{attribute 'reflection'} 
// Providing the event logger
FUNCTION_BLOCK FB_Event IMPLEMENTS I_Event
VAR_INPUT
	iLogger:					I_Logger;		// Interface has to be attached to a Valid target
END_VAR
VAR
    {attribute 'hide'} 
    {attribute 'instance-path'} 
    {attribute 'noinit'} 
    sInstancePath:				STRING(255);
	fbSymbolInfo: 				PLC_ReadSymInfoByNameEx;
	fbSystemTime: 				FB_LocalSystemTime;
	fbArguments:				FB_Argument;	
	fbVerbose:					FB_Message;
	fbInfo:						FB_Message;
	fbWarning:					FB_Message;
	fbError:					FB_Message;
	fbCritical:					FB_Message;
END_VAR
VAR_STAT
	nCycleTime:					UDINT;
	nTimestamp:					Tc2_Utilities.T_FILETIME64;		
END_VAR
(*
    Tc3_Event – TwinCAT 3 Event Logging Framework
    Copyright (c) Peter Zerlauth

    This component is provided under a Dual Licensing Model:

    1. GPLv3 Open-Source License
       - Free for personal, educational, and non-commercial use.
       - Commercial use allowed only if the entire application is published
         under GPLv3, including all modifications to this code.
       - Requires full disclosure of source code for derivative works.

    2. Commercial License
       - Required for integration into proprietary or closed-source products.
       - Removes all GPLv3 copyleft obligations.
       - Includes optional warranty, professional support, and long-term
         maintenance options.

    For commercial licensing, contact:
        info@peterzerlauth.com

    By using this Function Block you agree to the terms of the selected license.
*)

fbSymbolInfo();
IF nCycleTime <> TwinCAT_SystemInfoVarList._TaskInfo[GETCURTASKINDEXEX()].CycleTime THEN
	nCycleTime:= TwinCAT_SystemInfoVarList._TaskInfo[GETCURTASKINDEXEX()].CycleTime;
	fbSystemTime();
	nTimestamp:= SYSTEMTIME_TO_FILETIME64(fbSystemTime.systemTime);
	GVL.nTimestamp:= nTimestamp;	
END_IF

//FB_Init is always available implicitly and it is used primarily for initialization.
//The return value is not evaluated. For a specific influence, you can also declare the
//methods explicitly and provide additional code there with the standard initialization
//code. You can evaluate the return value.
METHOD FB_Init: BOOL
VAR_INPUT
    bInitRetains: BOOL; // TRUE: the retain variables are initialized (reset warm / reset cold)
    bInCopyCode: BOOL:= TRUE;  // TRUE: the instance will be copied to the copy code afterward (online change)   
END_VAR
fbSymbolInfo.SYMNAME:= F_InstancePath(sInstancePath);
fbSymbolInfo.PORT:= TwinCAT_SystemInfoVarList._AppInfo.AdsPort;
fbSymbolInfo.START:= TRUE;
fbSystemTime.bEnable:= TRUE;
END_METHOD

METHOD PUBLIC M_Critical : BOOL
VAR_INPUT
	sMessage:			STRING(255);
	nID:				UDINT;
END_VAR
VAR
	sArgument:			STRING;
	nPosition: 			INT;
END_VAR
IF sMessage = '' THEN
	RETURN;
END_IF

fbCritical.bActive:= TRUE;
fbCritical.sMessage:= sMessage;
fbCritical.eLogLevel:= E_LogLevel.Critical;
IF nID = 0 THEN
	fbCritical.nID:= F_Hash(sMessage);
ELSE
	fbCritical.nID:= nID;
END_IF
fbCritical.nTimestamp:= SYSTEMTIME_TO_FILETIME64(fbSystemTime.systemTime);
fbCritical.sArguments:= fbArguments.P_Value;
fbCritical.sDefault:= F_Print(sMessage, fbArguments.P_Value);
fbCritical.sSource:= fbSymbolInfo.SYMNAME;
fbCritical.sType:= fbSymbolInfo.SYMINFO.symDataType;

IF iLogger = 0 THEN
	F_Log(fbCritical);
ELSE
	iLogger.M_Log(fbCritical);
END_IF

	
fbArguments.M_Clear();
END_METHOD

METHOD PUBLIC M_Error : BOOL
VAR_INPUT
	sMessage:			STRING(255);
	nID:				UDINT;
END_VAR
VAR
	sArgument:			STRING;
	nPosition: 			INT;
END_VAR
IF sMessage = '' THEN
	RETURN;
END_IF

fbError.bActive:= TRUE;
fbError.sMessage:= sMessage;
fbError.eLogLevel:= E_LogLevel.Error;
IF nID = 0 THEN
	fbError.nID:= F_Hash(sMessage);
ELSE
	fbError.nID:= nID;
END_IF
fbError.nTimestamp:= SYSTEMTIME_TO_FILETIME64(fbSystemTime.systemTime);
fbError.sArguments:= fbArguments.P_Value;
fbError.sDefault:= F_Print(sMessage, fbArguments.P_Value);
fbError.sSource:= fbSymbolInfo.SYMNAME;
fbError.sType:= fbSymbolInfo.SYMINFO.symDataType;

IF iLogger = 0 THEN
	F_Log(fbError);
ELSE
	iLogger.M_Log(fbError);
END_IF

fbArguments.M_Clear();
END_METHOD

METHOD PUBLIC M_Info : BOOL
VAR_INPUT
	sMessage:			STRING(255);
	nID:				UDINT;
END_VAR
VAR
	sArgument:			STRING;
	nPosition: 			INT;
END_VAR
IF sMessage = '' THEN
	RETURN;
END_IF

fbInfo.bActive:= TRUE;
fbInfo.sMessage:= sMessage;
fbInfo.eLogLevel:= E_LogLevel.Info;
IF nID = 0 THEN
	fbInfo.nID:= F_Hash(sMessage);
ELSE
	fbInfo.nID:= nID;
END_IF
fbInfo.nTimestamp:= SYSTEMTIME_TO_FILETIME64(fbSystemTime.systemTime);
fbInfo.sArguments:= fbArguments.P_Value;
fbInfo.sDefault:= F_Print(sMessage, fbArguments.P_Value);
fbInfo.sSource:= fbSymbolInfo.SYMNAME;
fbInfo.sType:= fbSymbolInfo.SYMINFO.symDataType;

IF iLogger = 0 THEN
	F_Log(fbInfo);
ELSE
	iLogger.M_Log(fbInfo);
END_IF

fbArguments.M_Clear();
END_METHOD

METHOD M_Reset : BOOL
VAR_INPUT
END_VAR
VAR
	fbReset:					FB_Message;
END_VAR
fbReset.bActive:= TRUE;
fbReset.sMessage:= '###Reset###';
fbReset.eLogLevel:= E_LogLevel.Error;
fbReset.nID:= F_Hash(fbReset.sMessage);
fbReset.nTimestamp:= 0;
fbReset.sArguments:= '';
fbReset.sDefault:= '';
fbReset.sSource:= fbSymbolInfo.SYMNAME;
fbReset.sType:= fbSymbolInfo.SYMINFO.symDataType;

IF iLogger <> 0 THEN
	M_Reset:= iLogger.M_Log(fbReset);
END_IF
END_METHOD

METHOD PUBLIC M_Verbose : BOOL
VAR_INPUT
	sMessage:			STRING(255);		// content of the error message, placeholder %s
END_VAR
IF sMessage = '' THEN
	RETURN;
END_IF

fbVerbose.bActive:= TRUE;
fbVerbose.sMessage:= sMessage;
fbVerbose.eLogLevel:= E_LogLevel.Verbose;
fbVerbose.nID:= F_Hash(sMessage);
fbVerbose.nTimestamp:= SYSTEMTIME_TO_FILETIME64(fbSystemTime.systemTime);
fbVerbose.sArguments:= fbArguments.P_Value;
fbVerbose.sDefault:= F_Print(sMessage, fbArguments.P_Value);
fbVerbose.sSource:= fbSymbolInfo.SYMNAME;
fbVerbose.sType:= fbSymbolInfo.SYMINFO.symDataType;

IF iLogger = 0 THEN
	F_Log(fbVerbose);
ELSE
	iLogger.M_Log(fbVerbose);
END_IF


fbArguments.M_Clear();
END_METHOD

METHOD PUBLIC M_Warning : BOOL
VAR_INPUT
	sMessage:			STRING(255);
	nID:				UDINT;
END_VAR
IF sMessage = '' THEN
	RETURN;
END_IF

fbWarning.bActive:= TRUE;
fbWarning.sMessage:= sMessage;
fbWarning.eLogLevel:= E_LogLevel.Warning;
IF nID = 0 THEN
	fbWarning.nID:= F_Hash(sMessage);
ELSE
	fbWarning.nID:= nID;
END_IF
fbWarning.nTimestamp:= SYSTEMTIME_TO_FILETIME64(fbSystemTime.systemTime);
fbWarning.sArguments:= fbArguments.P_Value;
fbWarning.sDefault:= F_Print(sMessage, fbArguments.P_Value);
fbWarning.sSource:= fbSymbolInfo.SYMNAME;
fbWarning.sType:= fbSymbolInfo.SYMINFO.symDataType;

IF iLogger = 0 THEN
	F_Log(fbWarning);
ELSE
	iLogger.M_Log(fbWarning);
END_IF

fbArguments.M_Clear();
END_METHOD

PROPERTY PUBLIC P_Argument : I_Argument
GET
P_Argument:= fbArguments;
END_GET
END_PROPERTY

PROPERTY PUBLIC P_Logger : I_Logger
GET
P_Logger:= iLogger;
END_GET
SET
iLogger:= P_Logger;
END_SET
END_PROPERTY

END_FUNCTION_BLOCK

(* stored: Version 1.1.0.1
   POU FB_Event: Id {fcfa56ff-d0f1-4149-9de7-6f44354915c6}, SpecialFunc None
   Method FB_Init: Id {86bf7a82-ee08-4323-8f31-a4c33f4b211e}
   Method M_Critical: Id {7b4c91bf-8e3c-413c-a148-e271617106d9}
   Method M_Error: Id {11687e23-ea95-4e4f-aed4-4799ffa1ad84}
   Method M_Info: Id {7a920e55-da6d-473b-9aba-119c4de007e0}
   Method M_Reset: Id {3a4a22c9-fd2e-42d4-aaa7-202418505488}
   Method M_Verbose: Id {db95e385-16ed-493b-a6a5-28cc6625776b}
   Method M_Warning: Id {1aa0d3ef-0f74-4102-97d7-7d587822db85}
   Property P_Argument: Id {dd3bce54-33d7-4a6c-8d06-ad6a5d0ec566}
   Get Get: Id {9148b4be-b1fa-4fe4-a389-e96c939bba14}
   Property P_Logger: Id {98c079df-4944-4aae-a3d6-ca12ac41d1d4}
   Get Get: Id {7f49254e-94b6-4972-a1b5-02a92d10e780}
   Set Set: Id {4bbb606c-4053-49cc-ae04-84e1809ace25} *)
